FUNCTION_BLOCK Getriebemotor
VAR_INPUT
END_VAR
VAR_OUTPUT
END_VAR
VAR
END_VAR

END_FUNCTION_BLOCK

(* stored: Version 1.1.0.1, ProductVersion 3.1.4022.7
   POU Getriebemotor: Id {cb65ceda-4bf1-470d-b57d-3c08e6479214}, SpecialFunc None *)
